Omron CX-Programmer project NewProject (CX-Programmer 9.61)

# PLC NewPLC1: CP1E E20

## Global symbols (name address type ; comment)
0.00 BOOL  ; START
0.01 BOOL  ; STOP
0.02 BOOL  ; SENSOR 1
0.03 BOOL  ; SENSOR 2
0.04 BOOL  ; SENSOR 3
0.05 BOOL  ; SENSOR 4
100.00 BOOL  ; CONVEYOR
100.01 BOOL  ; Magazine
100.02 BOOL  ; INDIKATOR SENSOR 1
100.03 BOOL  ; INDIKATOR SENSOR 2
100.04 BOOL  ; INDIKATOR SENSOR 3

## Program NewProgram1 (cyclic task 0)

### Section Section1

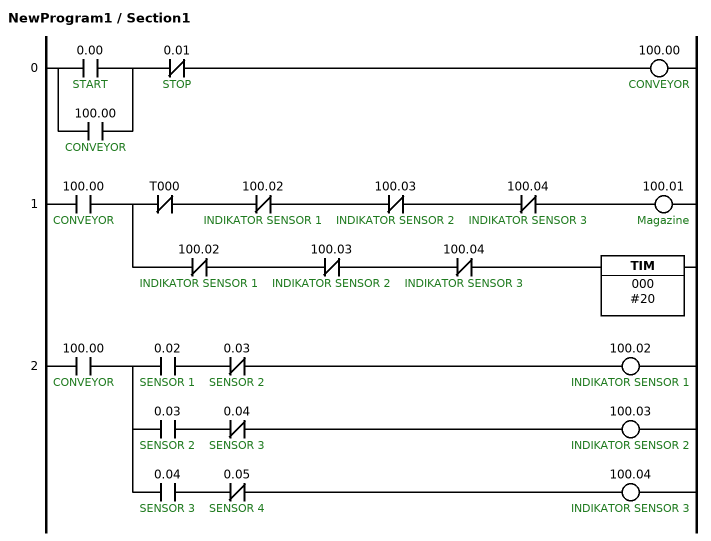
; rung 0
LD 0.00  ; START
OR 100.00  ; CONVEYOR
ANDNOT 0.01  ; STOP
OUT 100.00  ; CONVEYOR
; rung 1
LD 100.00  ; CONVEYOR
OUT TR0
ANDNOT T000
ANDNOT 100.02  ; INDIKATOR SENSOR 1
ANDNOT 100.03  ; INDIKATOR SENSOR 2
ANDNOT 100.04  ; INDIKATOR SENSOR 3
OUT 100.01  ; Magazine
LD TR0
ANDNOT 100.02  ; INDIKATOR SENSOR 1
ANDNOT 100.03  ; INDIKATOR SENSOR 2
ANDNOT 100.04  ; INDIKATOR SENSOR 3
TIM 000 #20
; rung 2
LD 100.00  ; CONVEYOR
OUT TR0
AND 0.02  ; SENSOR 1
ANDNOT 0.03  ; SENSOR 2
OUT 100.02  ; INDIKATOR SENSOR 1
LD TR0
AND 0.03  ; SENSOR 2
ANDNOT 0.04  ; SENSOR 3
OUT 100.03  ; INDIKATOR SENSOR 2
LD TR0
AND 0.04  ; SENSOR 3
ANDNOT 0.05  ; SENSOR 4
OUT 100.04  ; INDIKATOR SENSOR 3

### Section END
; rung 0
END(001)